{attribute 'qualified_only'}
{attribute 'strict'}
TYPE MAIN_STATE :
(
	STARTUP,
	IDLE,
	CHECK_TEST_READY,
	SET_TEST_VARIABLES,
	START_TEST,
	RUN_TEST,
	TEST_ERROR,
	TEST_COMPLETE,
	START_BLOWDOWN,
	BLOWDOWN,
	BLOWDOWN_COMPLETE,
	STOP,
	ESTOP,
	WAIT_FOR_RESET,
	RESETTING
);
END_TYPE

(* stored: Version 1.1.0.1, ProductVersion 3.1.4024.12
   EnumerationTextList MAIN_STATE: Id {d1b34753-8116-4e4e-b4f5-e3b219cd305a} *)
